(* PLC project Test, Beckhoff Automation GmbH TwinCAT PLC Control 3.5.10.30 *)
(* stored: creationDateTime 2017-11-09T14:50:50.6209258, modificationDateTime 2017-11-09T14:50:50.624425 *)

(* global variable list Labview *)
{attribute 'Tc2GvlVarNames'}
{attribute 'TcContextName':='PlcTaskStandard'}
VAR_GLOBAL	
	gui_ErrorMessages				:DINT;
	gui_Acknowledge					:BOOL;
	gui_Popup_VAR_AA				:STRING;	(*gui_Popup_VAR_AA :STRING;  (optional) Diese Variable enthält einen String welcher den String "VAR_AA" (Platzhalter) im Meldungstext ersetzt*)
	gui_ZustandMaschine				:INT;		(*0: Initialisierung, 1: Stopp, aber alles OK, 2: Produktion automatisch, 3: Schrittbetrieb, 4: Fehler, 5: Manuellbetrieb, 6: Notaus gedrückt, *)
	gui_UserLevel					:INT;		(*Opérateur, Réglage, Maintenance*)
	gui_UserLevelKeySwitchOn		:BOOL;		(*TRUE, wenn Schlüssel auf Service gedreht ist*)
	gui_AktPosAchseZ				:REAL;

END_VAR
